{attribute 'strict'}
TYPE E_VisuCtrUniversalMachineState :
(	
	VISU_CTRL_UNIVERSAL_MACHINE_WAIT_FOR_CMD	 	:= 0,	(*  *)
	VISU_CTRL_UNIVERSAL_MACHINE_INIT				:= 10,	(*  *)
	VISU_CTRL_UNIVERSAL_MACHINE_RESET				:= 20,	(*  *)
	VISU_CTRL_UNIVERSAL_MACHINE_START_AUTO			:= 30,	(*  *)
	VISU_CTRL_UNIVERSAL_MACHINE_STOP_AUTO			:= 40,	(*  *)
	VISU_CTRL_UNIVERSAL_MACHINE_SWITCH_TO_MANUAL	:= 50,	(*  *)
	VISU_CTRL_UNIVERSAL_MACHINE_SWITCH_TO_AUTO		:= 60,	(*  *)
	VISU_CTRL_UNIVERSAL_MACHINE_ABORT				:= -10	(*  *)
);
END_TYPE

(* stored: Version 1.1.0.1, ProductVersion 3.1.4024.12
   DUT E_VisuCtrUniversalMachineState: Id {dde2bbfa-fd86-4b36-b73d-7c9c8858e6ae} *)
